// TIA Portal V19 export
TYPE "MatCountHMI"
// stored: Access Published
   STRUCT
      PbFAKCalculation { ExternalVisible := 'False'; ExternalWritable := 'False'} : Bool;
      PbFAKDefault { ExternalVisible := 'False'; ExternalWritable := 'False'} : Bool;
      PbFAKPrevious { ExternalVisible := 'False'; ExternalWritable := 'False'} : Bool;
      FAKSetDefaultDone { ExternalVisible := 'False'; ExternalWritable := 'False'} : Bool;
      FAKCalcDone { ExternalVisible := 'False'; ExternalWritable := 'False'} : Bool;
      FAKSetPrevDone { ExternalVisible := 'False'; ExternalWritable := 'False'} : Bool;
      LenghtDesired { ExternalVisible := 'False'; ExternalWritable := 'False'} : LReal;
      LenghtMeasured { ExternalVisible := 'False'; ExternalWritable := 'False'} : LReal;
      FAKPrevious { ExternalVisible := 'False'; ExternalWritable := 'False'} : LReal;
   END_STRUCT;
END_TYPE
